// TIA Portal V18 export
VAR_GLOBAL   // PLC tag table "04 Costanti riordino quote"
   TempoInvioDatiPC AT %MD26 : Time;
   trasfincorso AT %M30.0 : Bool;
END_VAR
VAR_GLOBAL CONSTANT   // user constants
   NumRigheProduzione : DInt := 10;
   NumQuotePunzonaturaStorico : DInt := 5;
   NumPunzonateArticolo : DInt := 50;
   NumMaxPezziProfila : DInt := 80;
   NumQuotePunzonatura : DInt := 70;
   LunghezzaBanco : LReal := 1000.0;
END_VAR
